PROGRAM MAIN
VAR
	RampControlCycles	:	RampControlCycles;
	RampControlTime		:	RampControlTimers;
	StartPb				: 	BOOL;
	StopPb				: 	BOOL;
END_VAR

RampControlCycles(Start:= StartPb,
			Stop := StopPb,
			RampUpTime := 15,
			ContDutyTime := 20,
			RampDownTime := 5,
			RampMinVal := 10,
			RampMaxVal := 100,
			PlcCycleTimeMs := 10);
			
			
RampControlTime(Start:= StartPb,
			Stop := StopPb,
			RampUpTime := 7,
			ContDutyTime := 10,
			RampDownTime := 5,
			RampMinVal := 5,
			RampMaxVal := 70,
			PlcCycleTimeMs := 10);

END_PROGRAM

(* stored: Version 1.1.0.1, ProductVersion 3.1.4024.15
   POU MAIN: Id {4c63616b-78bd-4999-acc9-ad9d8ed1d662}, SpecialFunc None *)
